Staubli VAL3: start.pgx

program start()
begin
  call InitVariables()
  taskCreate "PositionUpdate",10,PositionUpdate()
  taskCreateSync "Communication",0.001,bOverrun,Communication()
  call InitInterface()
  call Deplacements()
end
